{attribute 'GeneratedUsingTerminal: EL2521-0124-0018'}
{attribute addProperty BoxType "EL2521-0124-0018"}
{attribute addProperty Id "PLS_EnabledBOOL1Status_of_outputBOOL1Sync_errorBOOL1TxPDO_ToggleBOOL1"}
{attribute addProperty CRC "1888949598"}
{attribute addProperty Size "4"}
TYPE Status_7097155E :
STRUCT
	{attribute addProperty Name "PLS_Enabled"}
	PLS_Enabled : BOOL;
	{attribute addProperty Name "Status_of_output"}
	Status_of_output : BOOL;
	{attribute addProperty Name "Sync_error"}
	Sync_error : BOOL;
	{attribute addProperty Name "TxPDO_Toggle"}
	TxPDO_Toggle : BOOL;
END_STRUCT
END_TYPE

(* stored: Version 1.2.0.0, ProductVersion 3.1.4024.9
   DUT Status_7097155E: Id {ba164ee8-3f9a-4b1f-9f83-db0be28d8fa3} *)
